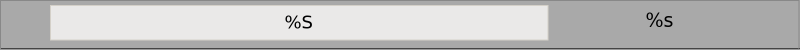
VISUALIZATION TOP  // 800x50
    Line (0,48) (800,48)
    Textfield (526,1 267x39), "%s", text variable: GVL_EHS.dtActTime
    Textfield (50,5 498x35), "%S", text variable: GVL_HMI.sMode
END_VISUALIZATION

(* stored: Version 1.1.0.1, ProductVersion 3.1.4024.15
   Visu TOP: Id {fb8a8d9c-6b00-4056-a0c4-2482275a17d0} *)
